PROGRAM Axis_05_Logic
VAR
	TON_0: TON;
	TON_1: TON;
	TON_2: TON;
	TON_3: TON;
	Axis_05_Velocity_Range: LREAL;
	Axis_05_Velocity_Scale: LREAL;
	Axis_05_Velocity_Raw: LREAL;
	Axis_05_Soft_Range: LREAL;
	Axis_05_Soft_Position: LREAL;
	Axis_05_Soft_Position_In_Range: LREAL;
END_VAR

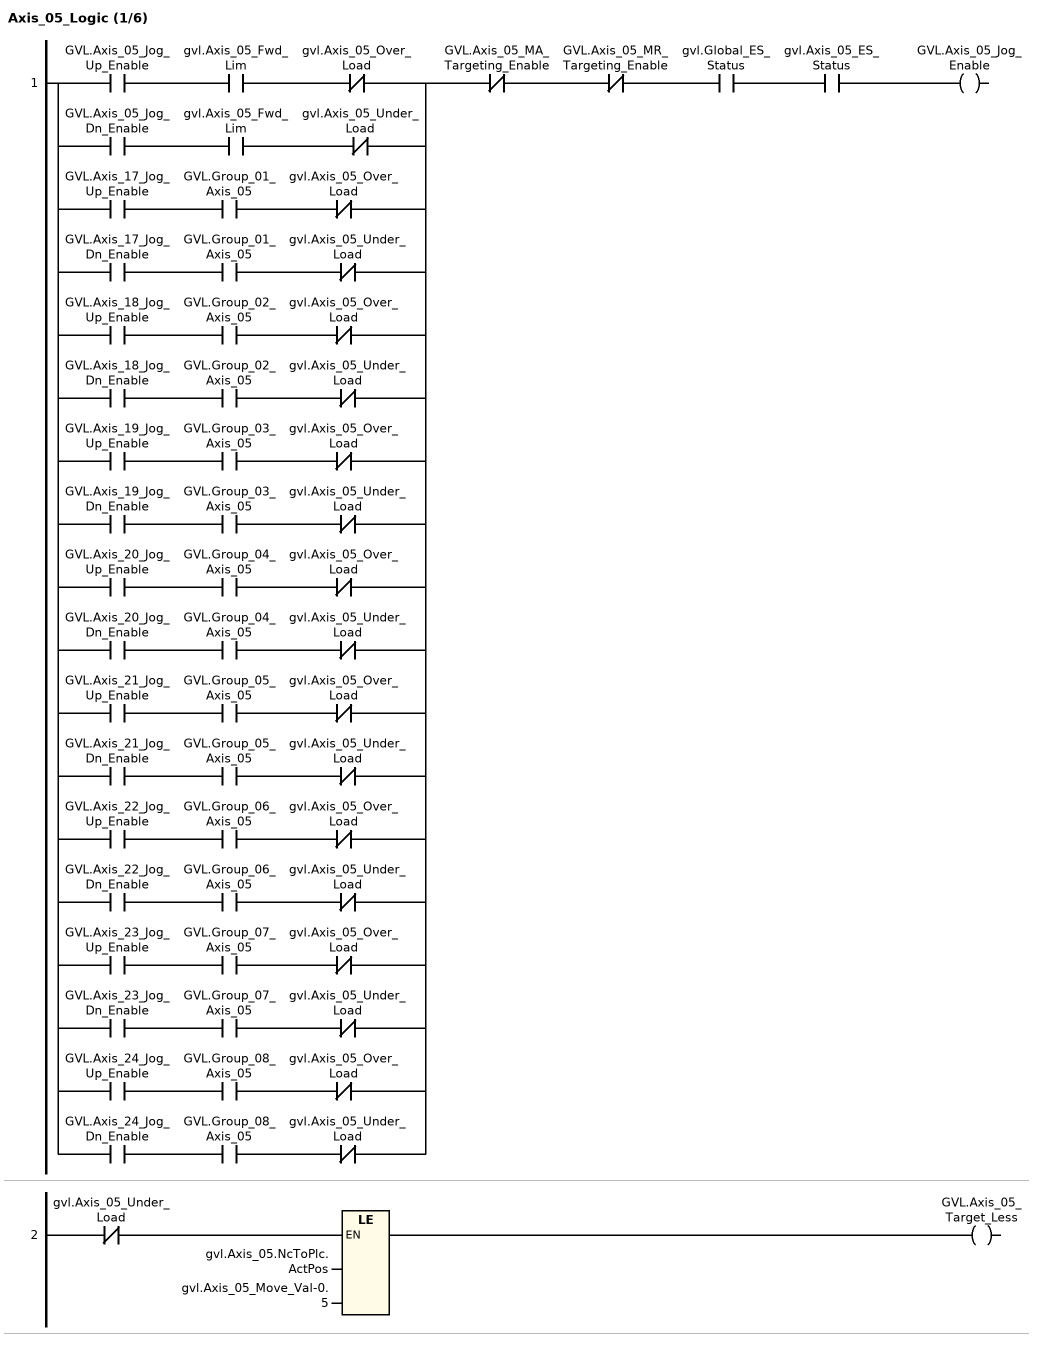
// NETWORK 1
GVL.Axis_05_Jog_Enable := (GVL.Axis_05_Jog_Up_Enable AND gvl.Axis_05_Fwd_Lim AND NOT gvl.Axis_05_Over_Load OR GVL.Axis_05_Jog_Dn_Enable AND gvl.Axis_05_Fwd_Lim AND NOT gvl.Axis_05_Under_Load OR GVL.Axis_17_Jog_Up_Enable AND GVL.Group_01_Axis_05 AND NOT gvl.Axis_05_Over_Load OR GVL.Axis_17_Jog_Dn_Enable AND GVL.Group_01_Axis_05 AND NOT gvl.Axis_05_Under_Load OR GVL.Axis_18_Jog_Up_Enable AND GVL.Group_02_Axis_05 AND NOT gvl.Axis_05_Over_Load OR GVL.Axis_18_Jog_Dn_Enable AND GVL.Group_02_Axis_05 AND NOT gvl.Axis_05_Under_Load OR GVL.Axis_19_Jog_Up_Enable AND GVL.Group_03_Axis_05 AND NOT gvl.Axis_05_Over_Load OR GVL.Axis_19_Jog_Dn_Enable AND GVL.Group_03_Axis_05 AND NOT gvl.Axis_05_Under_Load OR GVL.Axis_20_Jog_Up_Enable AND GVL.Group_04_Axis_05 AND NOT gvl.Axis_05_Over_Load OR GVL.Axis_20_Jog_Dn_Enable AND GVL.Group_04_Axis_05 AND NOT gvl.Axis_05_Under_Load OR GVL.Axis_21_Jog_Up_Enable AND GVL.Group_05_Axis_05 AND NOT gvl.Axis_05_Over_Load OR GVL.Axis_21_Jog_Dn_Enable AND GVL.Group_05_Axis_05 AND NOT gvl.Axis_05_Under_Load OR GVL.Axis_22_Jog_Up_Enable AND GVL.Group_06_Axis_05 AND NOT gvl.Axis_05_Over_Load OR GVL.Axis_22_Jog_Dn_Enable AND GVL.Group_06_Axis_05 AND NOT gvl.Axis_05_Under_Load OR GVL.Axis_23_Jog_Up_Enable AND GVL.Group_07_Axis_05 AND NOT gvl.Axis_05_Over_Load OR GVL.Axis_23_Jog_Dn_Enable AND GVL.Group_07_Axis_05 AND NOT gvl.Axis_05_Under_Load OR GVL.Axis_24_Jog_Up_Enable AND GVL.Group_08_Axis_05 AND NOT gvl.Axis_05_Over_Load OR GVL.Axis_24_Jog_Dn_Enable AND GVL.Group_08_Axis_05 AND NOT gvl.Axis_05_Under_Load) AND NOT GVL.Axis_05_MA_Targeting_Enable AND NOT GVL.Axis_05_MR_Targeting_Enable AND gvl.Global_ES_Status AND gvl.Axis_05_ES_Status;

// NETWORK 2
GVL.Axis_05_Target_Less := NOT gvl.Axis_05_Under_Load AND gvl.Axis_05.NcToPlc.ActPos <= (gvl.Axis_05_Move_Val-0.5);

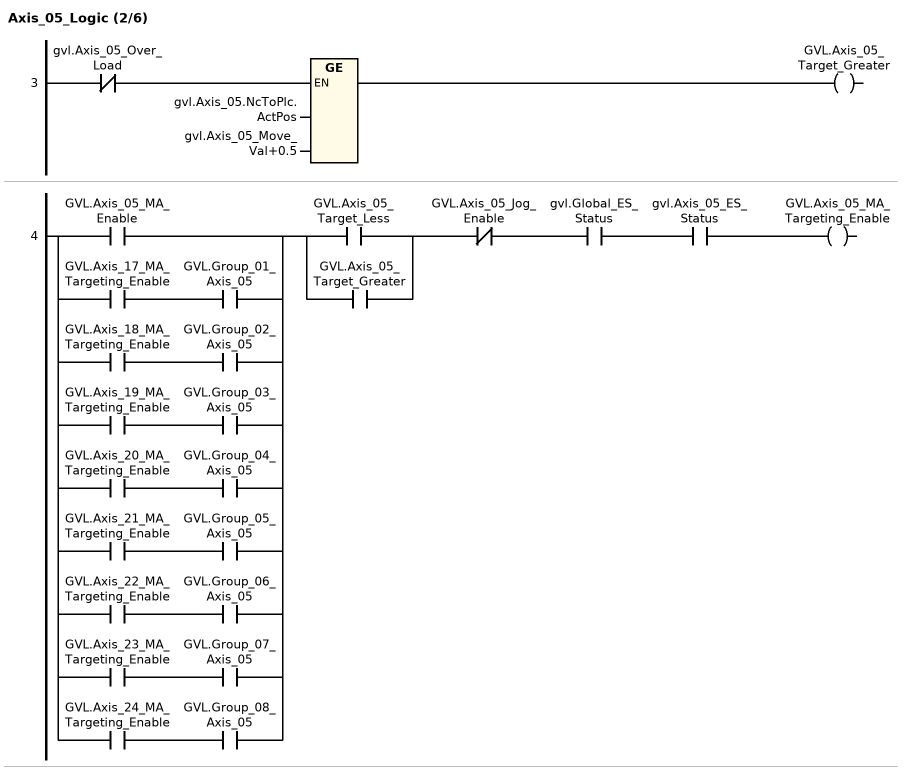
// NETWORK 3
GVL.Axis_05_Target_Greater := NOT gvl.Axis_05_Over_Load AND gvl.Axis_05.NcToPlc.ActPos >= (gvl.Axis_05_Move_Val+0.5);

// NETWORK 4
GVL.Axis_05_MA_Targeting_Enable := (GVL.Axis_05_MA_Enable OR GVL.Axis_17_MA_Targeting_Enable AND GVL.Group_01_Axis_05 OR GVL.Axis_18_MA_Targeting_Enable AND GVL.Group_02_Axis_05 OR GVL.Axis_19_MA_Targeting_Enable AND GVL.Group_03_Axis_05 OR GVL.Axis_20_MA_Targeting_Enable AND GVL.Group_04_Axis_05 OR GVL.Axis_21_MA_Targeting_Enable AND GVL.Group_05_Axis_05 OR GVL.Axis_22_MA_Targeting_Enable AND GVL.Group_06_Axis_05 OR GVL.Axis_23_MA_Targeting_Enable AND GVL.Group_07_Axis_05 OR GVL.Axis_24_MA_Targeting_Enable AND GVL.Group_08_Axis_05) AND (GVL.Axis_05_Target_Less OR GVL.Axis_05_Target_Greater) AND NOT GVL.Axis_05_Jog_Enable AND gvl.Global_ES_Status AND gvl.Axis_05_ES_Status;

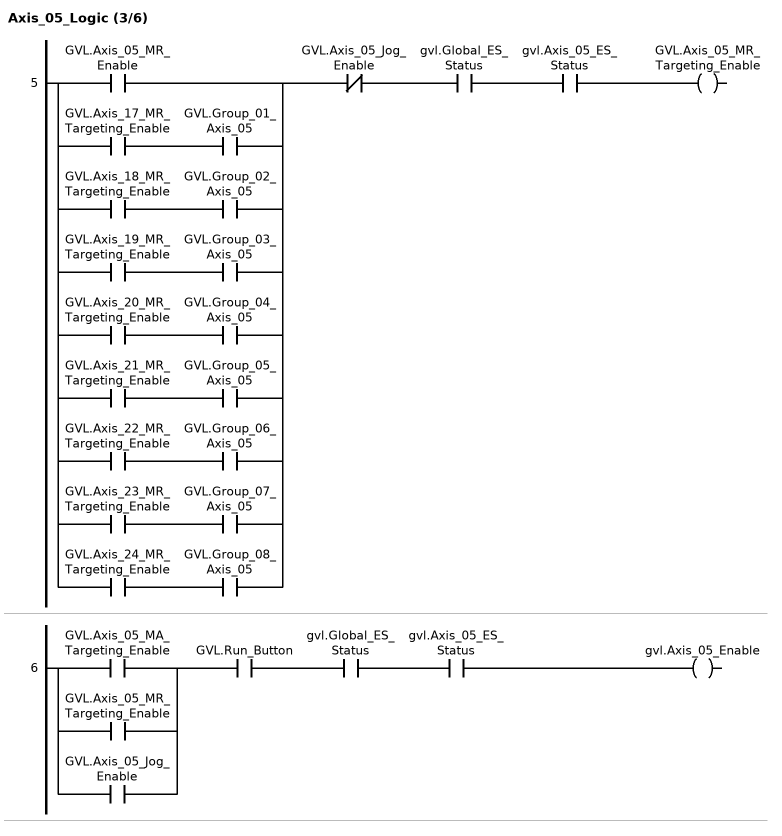
// NETWORK 5
GVL.Axis_05_MR_Targeting_Enable := (GVL.Axis_05_MR_Enable OR GVL.Axis_17_MR_Targeting_Enable AND GVL.Group_01_Axis_05 OR GVL.Axis_18_MR_Targeting_Enable AND GVL.Group_02_Axis_05 OR GVL.Axis_19_MR_Targeting_Enable AND GVL.Group_03_Axis_05 OR GVL.Axis_20_MR_Targeting_Enable AND GVL.Group_04_Axis_05 OR GVL.Axis_21_MR_Targeting_Enable AND GVL.Group_05_Axis_05 OR GVL.Axis_22_MR_Targeting_Enable AND GVL.Group_06_Axis_05 OR GVL.Axis_23_MR_Targeting_Enable AND GVL.Group_07_Axis_05 OR GVL.Axis_24_MR_Targeting_Enable AND GVL.Group_08_Axis_05) AND NOT GVL.Axis_05_Jog_Enable AND gvl.Global_ES_Status AND gvl.Axis_05_ES_Status;

// NETWORK 6
gvl.Axis_05_Enable := (GVL.Axis_05_MA_Targeting_Enable OR GVL.Axis_05_MR_Targeting_Enable OR GVL.Axis_05_Jog_Enable) AND GVL.Run_Button AND gvl.Global_ES_Status AND gvl.Axis_05_ES_Status;

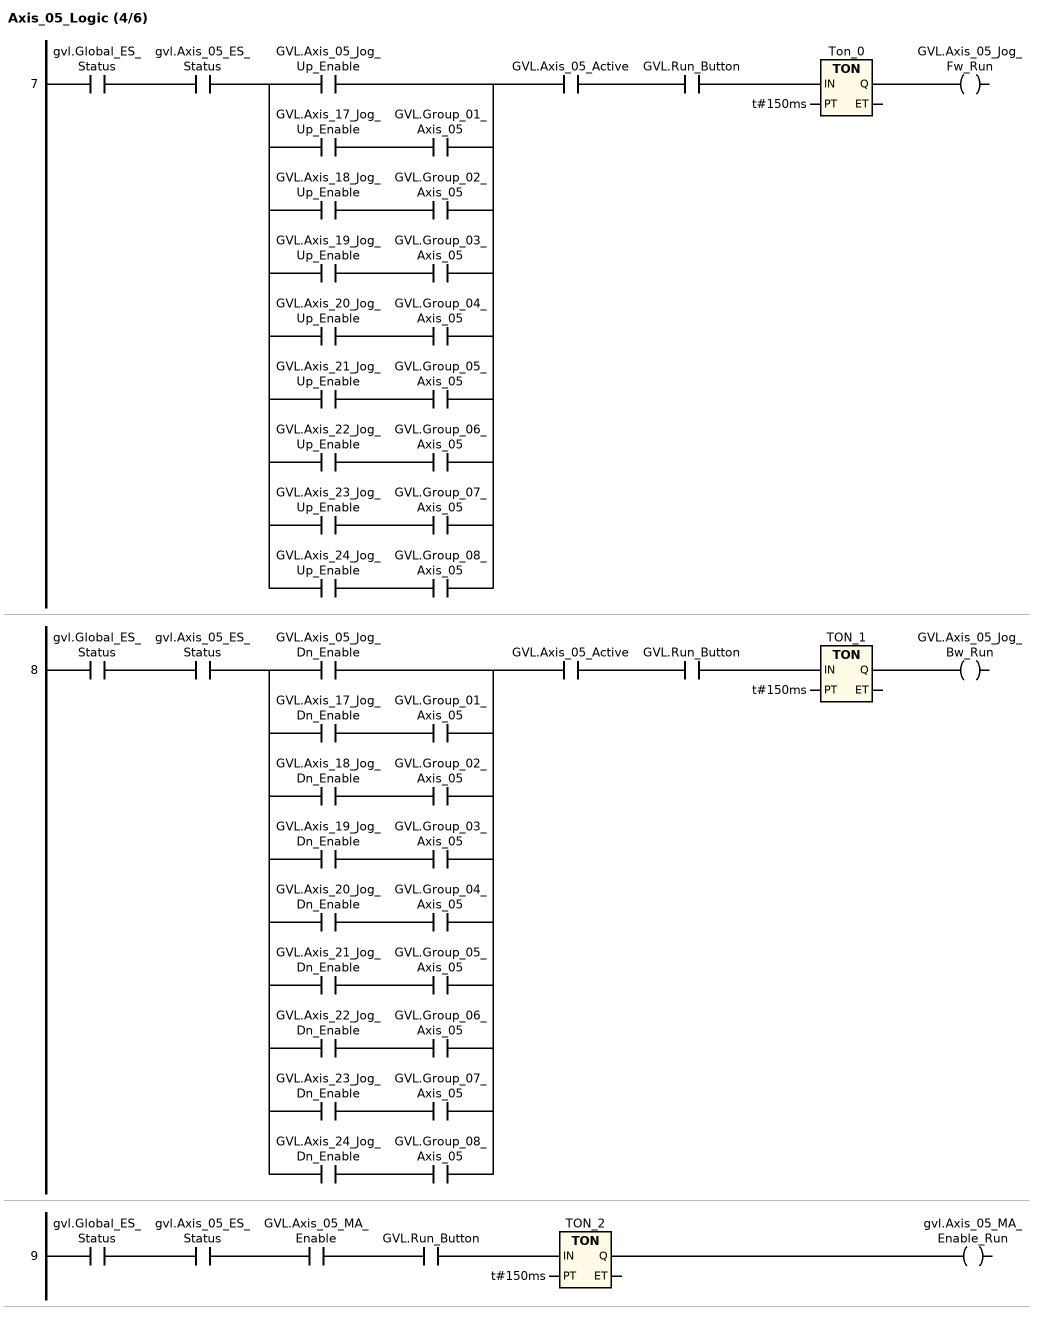
// NETWORK 7
Ton_0(IN := gvl.Global_ES_Status AND gvl.Axis_05_ES_Status AND (GVL.Axis_05_Jog_Up_Enable OR GVL.Axis_17_Jog_Up_Enable AND GVL.Group_01_Axis_05 OR GVL.Axis_18_Jog_Up_Enable AND GVL.Group_02_Axis_05 OR GVL.Axis_19_Jog_Up_Enable AND GVL.Group_03_Axis_05 OR GVL.Axis_20_Jog_Up_Enable AND GVL.Group_04_Axis_05 OR GVL.Axis_21_Jog_Up_Enable AND GVL.Group_05_Axis_05 OR GVL.Axis_22_Jog_Up_Enable AND GVL.Group_06_Axis_05 OR GVL.Axis_23_Jog_Up_Enable AND GVL.Group_07_Axis_05 OR GVL.Axis_24_Jog_Up_Enable AND GVL.Group_08_Axis_05) AND GVL.Axis_05_Active AND GVL.Run_Button, PT := t#150ms); // TON
GVL.Axis_05_Jog_Fw_Run := Ton_0.Q;

// NETWORK 8
TON_1(IN := gvl.Global_ES_Status AND gvl.Axis_05_ES_Status AND (GVL.Axis_05_Jog_Dn_Enable OR GVL.Axis_17_Jog_Dn_Enable AND GVL.Group_01_Axis_05 OR GVL.Axis_18_Jog_Dn_Enable AND GVL.Group_02_Axis_05 OR GVL.Axis_19_Jog_Dn_Enable AND GVL.Group_03_Axis_05 OR GVL.Axis_20_Jog_Dn_Enable AND GVL.Group_04_Axis_05 OR GVL.Axis_21_Jog_Dn_Enable AND GVL.Group_05_Axis_05 OR GVL.Axis_22_Jog_Dn_Enable AND GVL.Group_06_Axis_05 OR GVL.Axis_23_Jog_Dn_Enable AND GVL.Group_07_Axis_05 OR GVL.Axis_24_Jog_Dn_Enable AND GVL.Group_08_Axis_05) AND GVL.Axis_05_Active AND GVL.Run_Button, PT := t#150ms); // TON
GVL.Axis_05_Jog_Bw_Run := TON_1.Q;

// NETWORK 9
TON_2(IN := gvl.Global_ES_Status AND gvl.Axis_05_ES_Status AND GVL.Axis_05_MA_Enable AND GVL.Run_Button, PT := t#150ms); // TON
gvl.Axis_05_MA_Enable_Run := TON_2.Q;

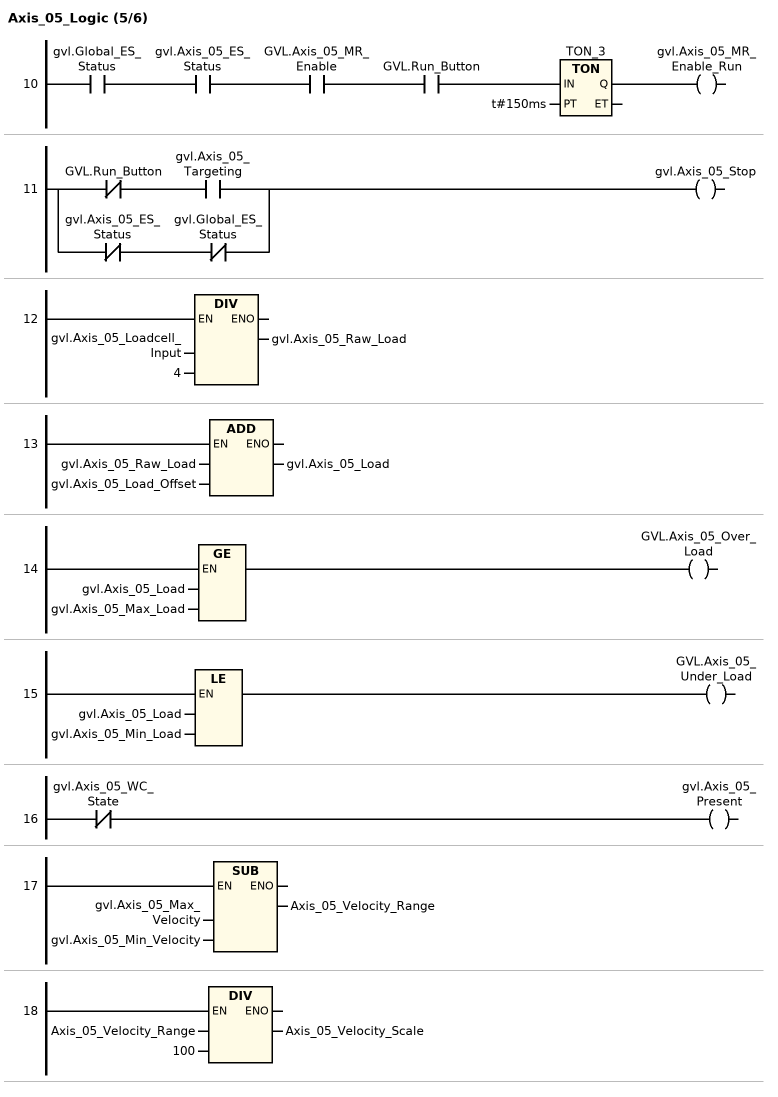
// NETWORK 10
TON_3(IN := gvl.Global_ES_Status AND gvl.Axis_05_ES_Status AND GVL.Axis_05_MR_Enable AND GVL.Run_Button, PT := t#150ms); // TON
gvl.Axis_05_MR_Enable_Run := TON_3.Q;

// NETWORK 11
gvl.Axis_05_Stop := NOT GVL.Run_Button AND gvl.Axis_05_Targeting OR NOT gvl.Axis_05_ES_Status AND NOT gvl.Global_ES_Status;

// NETWORK 12
gvl.Axis_05_Raw_Load := gvl.Axis_05_Loadcell_Input / 4;

// NETWORK 13
gvl.Axis_05_Load := gvl.Axis_05_Raw_Load + gvl.Axis_05_Load_Offset;

// NETWORK 14
GVL.Axis_05_Over_Load := gvl.Axis_05_Load >= gvl.Axis_05_Max_Load;

// NETWORK 15
GVL.Axis_05_Under_Load := gvl.Axis_05_Load <= gvl.Axis_05_Min_Load;

// NETWORK 16
gvl.Axis_05_Present := NOT gvl.Axis_05_WC_State;

// NETWORK 17
Axis_05_Velocity_Range := gvl.Axis_05_Max_Velocity - gvl.Axis_05_Min_Velocity;

// NETWORK 18
Axis_05_Velocity_Scale := Axis_05_Velocity_Range / 100;

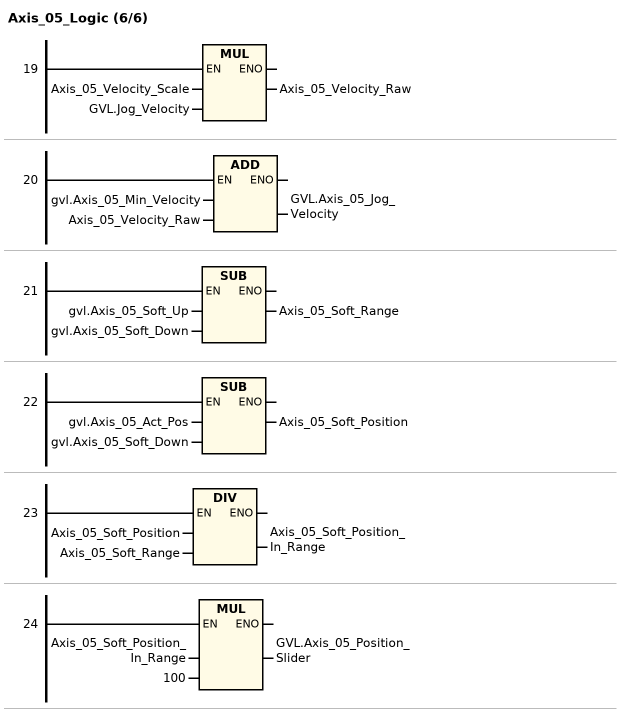
// NETWORK 19
Axis_05_Velocity_Raw := Axis_05_Velocity_Scale * GVL.Jog_Velocity;

// NETWORK 20
GVL.Axis_05_Jog_Velocity := gvl.Axis_05_Min_Velocity + Axis_05_Velocity_Raw;

// NETWORK 21
Axis_05_Soft_Range := gvl.Axis_05_Soft_Up - gvl.Axis_05_Soft_Down;

// NETWORK 22
Axis_05_Soft_Position := gvl.Axis_05_Act_Pos - gvl.Axis_05_Soft_Down;

// NETWORK 23
Axis_05_Soft_Position_In_Range := Axis_05_Soft_Position / Axis_05_Soft_Range;

// NETWORK 24
GVL.Axis_05_Position_Slider := Axis_05_Soft_Position_In_Range * 100;

END_PROGRAM

(* stored: Version 1.1.0.1, ProductVersion 3.1.4022.12
   POU Axis_05_Logic: Id {03e3346f-a92d-42f6-88e2-d2459a165ef1}, SpecialFunc None *)
